PROGRAM MAIN
VAR
END_VAR

END_PROGRAM

(* stored: Version 1.1.0.1, ProductVersion 3.1.4024.15
   POU MAIN: Id {4229cc46-d533-48cd-b8d1-1a73874c9d88}, SpecialFunc None *)
